// TIA Portal V20 export
DATA_BLOCK "BA030AZSCDR8_CathodeMainPnp2AxisX"   // DB147, Motion_DB
{ DB_Accessible_From_OPC_UA := 'FALSE' }
// stored: DBAccessibleFromOPCUA false, DBAccessibleFromWebserver false, InstanceOfName TO_SynchronousAxis, OfSystemLibElement TO_SynchronousAxis, OfSystemLibVersion 9.0
TO_SynchronousAxis   // technology object, version 9.0
// stored: Connection Interface Actor, InputAddress 42960, OutputAddress 42960
// stored: Connection Interface Sensor[1], InputAddress 42960, OutputAddress 42960, SensorIndexInActorTelegram 1
// stored: Connection Interface Torque, InputAddress 64560, OutputAddress 64560
// stored: SetPointCoupling Ref BA030A_MasterAxis, Type TO_SynchronousAxis
   // // inherited from TO_PositioningAxis
   // // inherited from TO_SpeedAxis
   // // inherited from TO_Axis
   // // inherited from TO_Object
   // VAR
   //    Actor : TO_Struct_Actor;
   //    DynamicLimits : TO_Struct_DynamicLimits;
   //    DynamicDefaults : TO_Struct_DynamicDefaults;
   // END_VAR
   // VAR
   //    Sensor : Array[1..4] of TO_Struct_Sensor;
   //    PositionLimits_HW : TO_Struct_PositionLimitsHW;
   //    Homing : TO_Struct_Homing;
   //    PositionControl : TO_Struct_PositionControl;
   // END_VAR
   // VAR
   //    SynchronizedMotion { S7_SetPoint := 'True'} : TO_Struct_SynchronizedMotion;
   //    StatusSynchronizedMotion { ExternalWritable := 'False'; S7_SetPoint := 'True'} : TO_Struct_StatusSynchronizedMotion;
   // END_VAR
BEGIN
   Actor.DataAdaption := 1;
   Actor.MotorType := 1;
   Actor.Interface.AddressIn.RID := 16#208072a;
   Actor.Interface.AddressIn.AREA := 16#81;
   Actor.Interface.AddressIn.OFFSET := 42960;
   Actor.Interface.AddressOut.RID := 16#208072b;
   Actor.Interface.AddressOut.AREA := 16#82;
   Actor.Interface.AddressOut.OFFSET := 42960;
   Actor.Interface.EnableTorqueData := true;
   Actor.Interface.TorqueDataAddressIn.RID := 16#2080742;
   Actor.Interface.TorqueDataAddressIn.AREA := 16#81;
   Actor.Interface.TorqueDataAddressIn.OFFSET := 64560;
   Actor.Interface.TorqueDataAddressOut.RID := 16#2080743;
   Actor.Interface.TorqueDataAddressOut.AREA := 16#82;
   Actor.Interface.TorqueDataAddressOut.OFFSET := 64560;
   Actor.LinearMotorDriveParameter.ReferenceVelocity := 195.0;
   Actor.LinearMotorDriveParameter.MaxVelocity := 250.0;
   Actor.LinearMotorDriveParameter.ReferenceForce := 3773.4;
   DynamicLimits.MaxVelocity := 2500.0;
   DynamicLimits.MaxAcceleration := 50000.0;
   DynamicLimits.MaxDeceleration := 50000.0;
   DynamicLimits.MaxJerk := 1000000.0;
   DynamicDefaults.EmergencyDeceleration := 50000.0;
   Sensor[1]."Type" := 2;
   Sensor[1].System := 0;
   Sensor[1].DataAdaption := 1;
   Sensor[1].Interface.AddressIn.RID := 16#208072a;
   Sensor[1].Interface.AddressIn.AREA := 16#81;
   Sensor[1].Interface.AddressIn.OFFSET := 42960;
   Sensor[1].Interface.AddressOut.RID := 16#208072b;
   Sensor[1].Interface.AddressOut.AREA := 16#82;
   Sensor[1].Interface.AddressOut.OFFSET := 42960;
   Sensor[1].Parameter.Resolution := 0.002048;
   Sensor[1].ActiveHoming.Mode := 2;
   Sensor[1].ActiveHoming.DigitalInputAddress.RID := 16#2000001;
   Sensor[1].ActiveHoming.DigitalInputAddress.AREA := 16#81;
   Sensor[1].ActiveHoming.DigitalInputAddress.OFFSET := 8110;
   Sensor[1].ActiveHoming.SwitchLevel := false;
   Sensor[1].PassiveHoming.Mode := 2;
   Sensor[1].PassiveHoming.Direction := 1;
   Sensor[1].PassiveHoming.DigitalInputAddress.RID := 16#2000001;
   Sensor[1].PassiveHoming.DigitalInputAddress.AREA := 16#81;
   Sensor[1].PassiveHoming.DigitalInputAddress.OFFSET := 8106;
   PositionLimits_HW.Active := true;
   PositionLimits_HW.MinSwitchLevel := false;
   PositionLimits_HW.MinSwitchAddress.RID := 16#2000001;
   PositionLimits_HW.MinSwitchAddress.AREA := 16#81;
   PositionLimits_HW.MinSwitchAddress.OFFSET := 8102;
   PositionLimits_HW.MaxSwitchLevel := false;
   PositionLimits_HW.MaxSwitchAddress.RID := 16#2000001;
   PositionLimits_HW.MaxSwitchAddress.AREA := 16#81;
   PositionLimits_HW.MaxSwitchAddress.OFFSET := 8103;
   PositionLimits_HW.ApproachBehavior := 1;
   Homing.AutoReversal := true;
   Homing.ApproachDirection := true;
   Homing.ApproachVelocity := 10.0;
   Homing.ReferencingVelocity := 2.0;
   PositionControl.EnableDSC := true;
   Actor.Interface.EnableTorqueData := True;
   _Sensor[1].PassiveHoming.DigitalInputAddress := BA030AZSBK04.12;
   _Sensor[1].ActiveHoming.DigitalInputAddress := BA030AZSBK04.16;
   _PositionLimits_HW.MinSwitchAddress := BA030AZSBK04.06;
   _PositionLimits_HW.MaxSwitchAddress := BA030AZSBK04.07;
   _Actor.Interface.Telegram := 105;
   _Actor.DataAdaptionOffline := True;
   _Sensor[1].Interface.Telegram := 105;
   _Sensor[1].DataAdaptionOffline := True;
END_DATA_BLOCK
